FUNCTION_BLOCK WoodBunkEx EXTENDS SectionEx
VAR //references to objects imported from Hardware GVL - using references instead of VAR_EXTERNAL or direct access allows local renaming
	robotLeft, robotRight : REFERENCE TO Robot;
	
	stagingTableLeft, stagingTableRight : REFERENCE TO WoodBunkTable;
	magazineLeft, magazineRight: REFERENCE TO MaterialStorage;
	
	strapper : REFERENCE TO StrapMachine;
	
	insertionLeft, insertionRight : REFERENCE TO Insertion;
	insertionBottom : REFERENCE TO AirPiston;
	
	toolStorageLeft, toolStorageRight : REFERENCE TO A21ToolStorage;
END_VAR
VAR
	conveyorPos : REAL;
	
	insertionSlots : ARRAY[Surface.TOP..Surface.BOTTOM] OF STRING;
	
	materialsArr : POINTER TO PositionMaterials; //array of PositionMaterials
	currentPair : REFERENCE TO PositionMaterials;
	
	stagingMaterial : STRING; //ex: currentPair.left
	currentMaterial : STRING; //ex: WDS18_WDS20 --> WDS18, then WDS20
	
	stagingTemplateReady : BOOL;
	stagingTemplateLeft : WoodBunkTable;
	stagingTemplateRight : WoodBunkTable;
	
	step : (RUN_TO_POSITION, PUSH, RUN_TO_STRAP, STRAP, RELEASE, RESET);
	
	//for staging use
	stageSet : INT;	
	stageStepLeft, stageStepRight : INT;
	iStagingSlotLeft, iStagingSlotRight : INT;
	
	robotLeftOutputs, robotRightOutputs : ARRAY[1..50] OF INT;
END_VAR
VAR
	tempInspectionSuite : VisionSuite; //send/receive from TcpServer
	leftInspectionFrame, rightInspectionFrame : VisionFrame; //parsed from above
END_VAR
VAR CONSTANT
	leftCamera : INT := 1;
	rightCamera : INT := 2;
END_VAR

entryRefPos := conveyorPos;
exitRefPos := conveyorPos;

SUPER^();

CASE status OF
	SectionStatus.IDLE:
		//RETURN;
	
	SectionStatus.ALIGNING:
		//
		
	SectionStatus.ACTIVE:
		//
		
	SectionStatus.CLEARING:
		stagingTemplateReady := FALSE;
		
	SectionStatus.COMPLETE:	
		//
		
	-100:
		RETURN;
		
END_CASE

materialsArr := ADR(currentBundle.woodBunk);

loaded := 
	insertionSlots[Surface.TOP] = materialsArr[iPair].top AND
	insertionSlots[Surface.LEFT] = materialsArr[iPair].left AND
	insertionSlots[Surface.RIGHT] = materialsArr[iPair].right AND
	insertionSlots[Surface.BOTTOM] = materialsArr[iPair].bottom;
	
//bundle needs this section's materials, and either robot failed
IF usesProcess() AND NOT(robotLeft.operational AND robotRight.operational) THEN 

	currentBypass := TRUE;
	RETURN;
END_IF //otherwise, carry over bypass from prev section

stage();

METHOD changeRobotsEOAT : BOOL
VAR_INPUT
END_VAR
IF robotLeft.tool <> sectionID THEN
	MEMSET(ADR(robotLeftOutputs), 0, SIZEOF(robotLeftOutputs));
	robotLeftOutputs[1] := A21.TOOL_CHANGE_CHIPBOARD;
	robotLeft.setParamsAndWait(robotLeftOutputs);
END_IF

IF robotRight.tool <> sectionID THEN
	MEMSET(ADR(robotRightOutputs), 0, SIZEOF(robotRightOutputs));
	robotRightOutputs[1] := A21.TOOL_CHANGE_CHIPBOARD;
	robotRight.setParamsAndWait(robotRightOutputs);
END_IF

changeRobotsEOAT := robotLeft.tool = sectionID AND robotRight.tool = sectionID;
END_METHOD

METHOD PROTECTED createStagingTemplate : BOOL
VAR
	remainingMaterial : STRING;
	splitMaterial : STRING;
	
	i : INT;
END_VAR
FOR i:=0 TO GVL.maxPairs BY 1 DO //iterate through all pairs and autofill the template
	//LEFT TABLE
	remainingMaterial := materialsArr[i].top;
	WHILE FIND(remainingMaterial, '_') > 0 DO //until no underscore found
		splitCombinedMaterials(remainingMaterial, splitMaterial);
		stagingTemplateLeft.autofill(splitMaterial);
	END_WHILE
	stagingTemplateLeft.autofill(remainingMaterial);
	
	remainingMaterial := materialsArr[i].left;
	WHILE FIND(remainingMaterial, '_') > 0 DO
		splitCombinedMaterials(remainingMaterial, splitMaterial);
		stagingTemplateLeft.autofill(splitMaterial);
	END_WHILE
	stagingTemplateLeft.autofill(remainingMaterial);
	
	//RIGHT TABLE
	remainingMaterial := materialsArr[i].right;
	WHILE FIND(remainingMaterial, '_') > 0 DO
		splitCombinedMaterials(remainingMaterial, splitMaterial);
		stagingTemplateRight.autofill(splitMaterial);
	END_WHILE
	stagingTemplateRight.autofill(remainingMaterial);
	
	remainingMaterial := materialsArr[i].bottom;
	WHILE FIND(remainingMaterial, '_') > 0 DO
		splitCombinedMaterials(remainingMaterial, splitMaterial);
		stagingTemplateRight.autofill(splitMaterial);
	END_WHILE
	stagingTemplateRight.autofill(remainingMaterial);
END_FOR
END_METHOD

METHOD findOpenSlot : BOOL
VAR_INPUT
	materialCode : STRING;
END_VAR
VAR_OUTPUT
	openSlot : INT := 0;
END_VAR
(*
IF FIND(materialCode, 'WDW') > 0 THEN //top wide, load in slot 0-1
	FOR i:=1 TO 2 BY 1 DO
		IF stageTableLeft[i] = '' THEN
			findOpenSlot := TRUE;
			openSlot := i;
			RETURN;
		END_IF
	END_FOR
	
ELSIF FIND(materialCode, 'WDT') > 0 OR FIND(materialCode, 'WDS') > 0 THEN //top std and sides, load in slot 2-9
	FOR i:=3 TO 10 BY 1 DO
		IF stageTableLeft[i] = '' THEN
			findOpenSlot := TRUE;
			openSlot := i;
			RETURN;
		END_IF
	END_FOR
	
END_IF
*)
END_METHOD

METHOD initHardware : BOOL
conveyors := ADR(allConveyors);

robotLeft REF= robots[1];
robotRight REF= robots[2];

strapper REF= strapperA21;

insertionLeft REF= insertionA21Left;
insertionLeft REF= insertionA21Right;

stagingTableLeft REF= stagingTableLeft;
stagingTableRight REF= stagingTableRight;

magazineLeft REF= woodBunkMagazineLeft;
magazineRight REF= woodBunkMagazineRight;

(*
strapper REF= Hardware.strapper;

insertionLeft REF= Hardware.insertionWoodBunkSides[Surface.LEFT];
insertionLeft REF= Hardware.insertionWoodBunkSides[Surface.RIGHT];

stagingTableLeft REF= Hardware.stagingTable[Surface.LEFT];
stagingTableRight REF= Hardware.stagingTable[Surface.RIGHT];

magazineLeft REF= Hardware.woodBunkMagazine[Surface.LEFT];
magazineRight REF= Hardware.woodBunkMagazine[Surface.RIGHT];
*)
END_METHOD

METHOD PROTECTED load : BOOL
VAR_INPUT
	pair : REFERENCE TO PositionMaterials;
END_VAR
IF NOT robotLeft.operational OR NOT robotLeft.operational THEN
	error := TRUE;
	
	currentBypass := TRUE;
	RETURN;
END_IF

IF NOT (robotLeft.reserve(sectionID) AND robotRight.reserve(sectionID)) THEN
	RETURN;
END_IF

IF NOT (robotLeft.tool = sectionID AND robotRight.tool = sectionID) THEN //robots have wrong tool
	changeRobotsEOAT(); //wait for robots to finish changing tools
	RETURN;
END_IF


CASE loadSet OF
	0: //top and bottom
		IF 
			loadingSequence(
				actingRobot:= robotLeft, 
				robotOutputs:= robotLeftOutputs, 
				stagingTable:= stagingTableLeft, 
				loadStep:= loadStepLeft, 
				surfaceID:= Surface.TOP, 
				material:= pair.top, 
				fail=> )
			AND
			loadingSequence(
				actingRobot:= robotRight, 
				robotOutputs:= robotRightOutputs, 
				stagingTable:= stagingTableRight, 
				loadStep:= loadStepRight, 
				surfaceID:= Surface.BOTTOM, 
				material:= pair.bottom, 
				fail=> )
		THEN
			loadStepLeft := loadStepRight := 0;
			loadSet := 10;
		END_IF
		
	10: //sides
		IF
			loadingSequence(
				actingRobot:= robotLeft, 
				robotOutputs:= robotLeftOutputs, 
				stagingTable:= stagingTableLeft, 
				loadStep:= loadStepLeft, 
				surfaceID:= Surface.LEFT, 
				material:= pair.left, 
				fail=> )
			AND
			loadingSequence(
				actingRobot:= robotRight, 
				robotOutputs:= robotRightOutputs, 
				stagingTable:= stagingTableRight, 
				loadStep:= loadStepRight, 
				surfaceID:= Surface.RIGHT, 
				material:= pair.right, 
				fail=> )
		THEN
			loadStepLeft := loadStepRight := 0;
			loadSet := COMPLETE;
		END_IF
		
	COMPLETE:
		loadSet := 0;
		loadStepLeft := loadStepRight := 0;
		
		loaded := 
			insertionSlots[Surface.TOP] = materialsArr[iPair].top AND
			insertionSlots[Surface.LEFT] = materialsArr[iPair].left AND
			insertionSlots[Surface.RIGHT] = materialsArr[iPair].right AND
			insertionSlots[Surface.BOTTOM] = materialsArr[iPair].bottom;
		
		robotLeft.release(sectionID);
		robotRight.release(sectionID);
		
		load := TRUE;
END_CASE
END_METHOD

METHOD loadBottom : BOOL
VAR_IN_OUT //acting refers to which robot is performing the task, if the designated robot fails the other may take over
	actingRobot : Robot;
	robotOutputs : ARRAY[1..50] OF INT;
	actingStagingTable : WoodBunkTable;
	actingLoadStep : INT;
END_VAR
VAR_INPUT
	material : STRING;
END_VAR
VAR_OUTPUT
	fail : BOOL;
END_VAR
VAR
	slot : INT;
END_VAR
IF
	actingLoadStep <> COMPLETE AND_THEN
	NOT actingRobot.reserve(sectionID)
THEN
	RETURN;
END_IF

CASE actingLoadStep OF
	0:
		IF NOT actingStagingTable.findSlot(materialID := material, atSlot => slot) THEN
			fail := TRUE;
			RETURN;
		END_IF
		
		MEMSET(ADR(robotOutputs), 0, SIZEOF(robotOutputs));
		robotOutputs[1] := A21.LOAD_BUNK_TO_BOTTOM;
		robotOutputs[2] := slot;
		
		IF actingRobot.setParamsAndWait(robotOutputs) THEN
			actingLoadStep := COMPLETE;
		END_IF
		
	COMPLETE:
		//turn suction on
		actingRobot.release(sectionID);
		loadBottom := TRUE;
END_CASE
END_METHOD

METHOD loadingSequence : BOOL
VAR_IN_OUT
	actingRobot : Robot;
	robotOutputs : ARRAY[1..50] OF INT;
	stagingTable : WoodBunkTable;
	loadStep : INT;
END_VAR
VAR_INPUT
	surfaceID : Surface;
	material : STRING;
END_VAR
VAR_OUTPUT
	fail : BOOL;
END_VAR
VAR
	slot : INT;
END_VAR
IF material = '' THEN
	loadingSequence := TRUE;
	RETURN;
END_IF

CASE loadStep OF
	0:
		IF NOT stagingTable.findSlot(materialID := material, atSlot => slot) THEN
			fail := TRUE;
			RETURN;
		END_IF
		
		MEMSET(ADR(robotOutputs), 0, SIZEOF(robotOutputs));
		CASE surfaceID OF
			Surface.TOP: 					robotOutputs[1] := A21.LOAD_BUNK_TO_TOP;
			Surface.LEFT, Surface.RIGHT: 	robotOutputs[1] := A21.LOAD_BUNK_TO_SIDE;
			Surface.BOTTOM: 				robotOutputs[1] := A21.LOAD_BUNK_TO_BOTTOM;
		END_CASE
		robotOutputs[2] := slot;
		
		IF actingRobot.setParamsAndWait(robotOutputs) THEN
			loadStep := COMPLETE;
		END_IF
		
	COMPLETE:
		//turn suction on
		actingRobot.release(sectionID);
		loadingSequence := TRUE;
		
END_CASE
END_METHOD

METHOD loadSides : BOOL
VAR_IN_OUT //acting refers to which robot is performing the task, if the designated robot fails the other may take over
	actingRobot : Robot;
	robotOutputs : ARRAY[1..50] OF INT;
	actingStagingTable : WoodBunkTable;
	actingLoadStep : INT;
END_VAR
VAR_INPUT
	material : STRING;
END_VAR
VAR_OUTPUT
	fail : BOOL;
END_VAR
VAR
	slot : INT;
END_VAR
IF
	actingLoadStep <> COMPLETE AND_THEN
	NOT actingRobot.reserve(sectionID)
THEN
	RETURN;
END_IF

CASE actingLoadStep OF
	0:
		IF NOT actingStagingTable.findSlot(materialID := material, atSlot => slot) THEN
			fail := TRUE;
			RETURN;
		END_IF
		
		MEMSET(ADR(robotOutputs), 0, SIZEOF(robotOutputs));
		robotOutputs[1] := A21.LOAD_BUNK_TO_SIDE;
		robotOutputs[2] := slot;
		
		IF actingRobot.setParamsAndWait(robotOutputs) THEN
			actingLoadStep := COMPLETE;
		END_IF
		
	COMPLETE:
		//turn suction on
		actingRobot.release(sectionID);
		loadSides := TRUE;
END_CASE
END_METHOD

METHOD loadTop : BOOL
VAR_IN_OUT //acting refers to which robot is performing the task, if the designated robot fails the other may take over
	actingRobot : Robot;
	robotOutputs : ARRAY[1..50] OF INT;
	actingStagingTable : WoodBunkTable;
	actingLoadStep : INT;
END_VAR
VAR_INPUT
	material : STRING;
END_VAR
VAR_OUTPUT
	fail : BOOL;
END_VAR
VAR
	slot : INT;
END_VAR
IF
	actingLoadStep <> COMPLETE AND_THEN
	NOT actingRobot.reserve(sectionID)
THEN
	RETURN;
END_IF

CASE actingLoadStep OF
	0:
		IF NOT actingStagingTable.findSlot(materialID := material, atSlot => slot) THEN
			fail := TRUE;
			RETURN;
		END_IF
		
		MEMSET(ADR(robotOutputs), 0, SIZEOF(robotOutputs));
		robotOutputs[1] := A21.LOAD_BUNK_TO_TOP;
		robotOutputs[2] := slot;
		
		IF actingRobot.setParamsAndWait(robotOutputs) THEN
			actingLoadStep := COMPLETE;
		END_IF
		
	COMPLETE:
		//turn suction on
		actingRobot.release(sectionID);
		loadTop := TRUE;
END_CASE
END_METHOD

METHOD PROTECTED process : BOOL
VAR
	currentPair : REFERENCE TO PositionMaterials REF= materialsArr[iPair];
END_VAR
IF iPair >= GVL.maxPairs THEN
	process := TRUE;
	RETURN;
END_IF

IF NOT PositionIsValid(pair:= currentPair) THEN
	step := 0;
	iPair := iPair + 1;
	RETURN;
END_IF

CASE step OF
	RUN_TO_POSITION: //free run until position reached
		IF directionCheckAndSet(conveyorPos, currentPair.position) AND load(pair:= currentPair) THEN
			step := PUSH;
		END_IF

	PUSH: //push command
		setConveyorMode(ConveyorMode.STOP);
		IF
			NOT insertionLeft.align(currentBundle.height/2) OR
			NOT insertionRight.align(currentBundle.height/2)
		THEN
			RETURN;
		END_IF
		
		insertionLeft.press();
		insertionRight.press();
		insertionBottom.extend();
		
		IF insertionLeft.contact AND insertionRight.contact AND insertionBottom.contact THEN		
			step := STRAP;
		END_IF
		
	STRAP: //strap command
		//turn off suction here
		setConveyorMode(ConveyorMode.STOP);
		IF strapper.ready OR (NOT strapper.busy AND NOT strapper.error) THEN
			strapper.strap();
		END_IF
		
		IF strapper.done THEN
			step := RELEASE;
		END_IF
		
	RELEASE: //release command
		setConveyorMode(ConveyorMode.STOP);
		
		IF NOT insertionLeft.home THEN
			insertionLeft.align(0);
			insertionLeft.release();
		END_IF
		
		IF NOT insertionRight.home THEN
			insertionRight.align(0);
			insertionRight.release();
		END_IF
		
		IF insertionLeft.home AND insertionRight.home THEN
			step := RESET;
		END_IF
		
	RESET: //reset
		setConveyorMode(ConveyorMode.FORWARD);
		iPair := iPair + 1;
		
		step := 0;
		
END_CASE
END_METHOD

METHOD splitCombinedMaterials : BOOL
VAR_IN_OUT
	materialID : STRING;
	splitMaterial : STRING;
END_VAR
VAR
	i : INT;
END_VAR
FindAndSplitChar(
	sSeparatorChar:= '_', 
	pSrcString:= ADR(materialID), 
	pLeftString:= ADR(splitMaterial), 
	nLeftSize:= SIZEOF(splitMaterial), 
	pRightString:= ADR(materialID), 
	nRightSize:= SIZEOF(materialID), 
	bSearchFromRight:= FALSE);
END_METHOD

METHOD stage : BOOL
//robot reservation needs to be constantly checked so it is not in the state machine
IF NOT (robotLeft.reserve(sectionID) AND robotRight.reserve(sectionID)) THEN
	RETURN;
END_IF

IF NOT (robotLeft.tool = sectionID AND robotRight.tool = sectionID) THEN //robots have wrong tool
	changeRobotsEOAT(); //wait for robots to finish changing tools
	RETURN;
END_IF

CASE stageSet OF
	0: //create staging template
		createStagingTemplate();
		stageSet := 10;
	
	10: //staging sequence
		IF TcpServer1Vision.fetch(tempInspectionSuite.data) THEN
			(*
				1 - parse
				2 - determine if the camera number is for left or right staging
				3 - copy into appropriate frame
			*)
			MEMCPY(
				ADR(tempInspectionSuite.json),
				ADR(tempInspectionSuite.data),
				MIN( SIZEOF(tempInspectionSuite.json), SIZEOF(tempInspectionSuite.data) ));
			
			VisionJsonParser(
				jsonString:= tempInspectionSuite.json,
				visionData=> );
			
			IF NOT FrameIsValid(tempInspectionSuite.frame) THEN
				//
			
			ELSIF tempInspectionSuite.frame.CameraNumber = leftCamera THEN
				leftInspectionFrame := tempInspectionSuite.frame;
				
			ELSIF tempInspectionSuite.frame.CameraNumber = rightCamera THEN
				rightInspectionFrame := tempInspectionSuite.frame;
				
			END_IF
		END_IF
		

		IF
			stagingSequence(
				template:= stagingTemplateLeft, 
				magazine:= magazineLeft, 
				table:= stagingTableLeft, 
				stagingSlot:= iStagingSlotLeft,
				actingRobot:= robotLeft, 
				robotOutputs:= robotLeftOutputs,
				inspectionFrame:= leftInspectionFrame, 
				actingStep:= stageStepLeft, 
				camera:= leftCamera, 
				fail=> )
			AND
			stagingSequence(
				template:= stagingTemplateRight, 
				magazine:= magazineRight, 
				table:= stagingTableRight, 
				stagingSlot:= iStagingSlotRight,
				actingRobot:= robotRight, 
				robotOutputs:= robotRightOutputs,
				inspectionFrame:= rightInspectionFrame, 
				actingStep:= stageStepRight, 
				camera:= rightCamera, 
				fail=> )
		THEN
			stageStepLeft := stageStepRight := 0;
			iStagingSlotLeft := iStagingSlotRight := 0;
			
			stageSet := COMPLETE;
		END_IF
		
	COMPLETE:
		stageSet := 0;
		stageStepLeft := stageStepRight := 0;
		
		robotLeft.release(sectionID);
		robotRight.release(sectionID);
		
		stage := TRUE;
		
END_CASE
END_METHOD

METHOD stageLeft : BOOL
VAR_IN_OUT
	template : WoodBunkTable;
	magazine : MaterialStorage;
	table : WoodBunkTable;
	actingStagingSlot : INT;
	actingRobot : Robot;
	robotOutputs : ARRAY[1..50] OF INT;
	actingFrame : VisionFrame;
	actingStep : INT;
END_VAR
VAR_INPUT
	camera : INT;
END_VAR
VAR_OUTPUT
	fail : BOOL;
END_VAR
VAR
	finished : BOOL;
	slot : INT;
	templateArr : POINTER TO STRING;
END_VAR
VAR CONSTANT
	WIP : INT := 0;
	PASSED : INT := 1;
	FAILED : INT := 2;
END_VAR
IF table.isFull() OR actingStagingSlot > 10 THEN
	stageLeft := TRUE;
	RETURN;
END_IF

templateArr := template.getSlotsAsArray();

//follow the template as is
IF NOT magazine.findSlot(materialID:= templateArr[actingStagingSlot], atSlot => slot) THEN
	fail := TRUE;
	RETURN;
END_IF

IF actingStep > 0 THEN
	finished := actingRobot.setCommandAndWait(A21.STAGE_BUNK, slot, actingStagingSlot, 0);
END_IF

CASE actingStep OF
	0: //command
		IF actingRobot.inputs[5].10 THEN
			actingStep := 10;
		END_IF
		
	10: //request inspection
		tempInspectionSuite.frame.MaterialID := templateArr[actingStagingSlot];
		tempInspectionSuite.frame.CheckFor := 'ORIENTATION';
		tempInspectionSuite.frame.CameraNumber := camera;
	
		CreateJsonDocumentAuto(
			visionFrameData:= tempInspectionSuite.frame, 
			jsonDocument=> tempInspectionSuite.json);
		
		MEMCPY(
			ADR(tempInspectionSuite.data), 
			ADR(tempInspectionSuite.json), 
			MIN( SIZEOF(tempInspectionSuite.data), SIZEOF(tempInspectionSuite.json) ));
			
		TcpServer1Vision.queue(tempInspectionSuite.data);
		
		actingStep := 20;
	
	20: //fetch inspection data and parse
		actingRobot.setCommandAndWait(A21.STAGE_BUNK, slot, actingStagingSlot, 0);
		robotOutputs[4] := 0;
		
		IF NOT FrameIsValid(actingFrame) THEN
			RETURN;
		END_IF
		
		IF actingFrame.SuccessFlag = 1 THEN
			robotOutputs[4] := PASSED;
		ELSE
			robotOutputs[4] := FAILED;
		END_IF
		actingStep := 30;
		
	30: //finish command
		IF finished THEN
			IF actingFrame.SuccessFlag = 1 THEN
				actingStagingSlot := actingStagingSlot + 1;
			END_IF
			
			actingStep := 0;
		END_IF
END_CASE
END_METHOD

METHOD stageRight : BOOL
VAR_IN_OUT
	template : WoodBunkTable;
	magazine : MaterialStorage;
	table : WoodBunkTable;
	actingStagingSlot : INT;
	actingRobot : Robot;
	actingFrame : VisionFrame;
	actingStep : INT;
END_VAR
VAR_INPUT
	camera : INT;
END_VAR
VAR_OUTPUT
	fail : BOOL;
END_VAR
VAR
	finished : BOOL;
	robotOutputs : POINTER TO INT;
	
	slot : INT;
	templateArr : POINTER TO STRING;
	
END_VAR
IF table.isFull() OR actingStagingSlot > 10 THEN
	stageRight := TRUE;
	RETURN;
END_IF

templateArr := template.getSlotsAsArray();

//follow the template as is
IF NOT magazine.findSlot(materialID:= templateArr[actingStagingSlot], atSlot => slot) THEN
	fail := TRUE;
	RETURN;
END_IF

IF actingStep > 0 THEN
	finished := actingRobot.setCommandAndWait(A21.STAGE_BUNK, slot, actingStagingSlot, 0);
END_IF

CASE actingStep OF
	0: //command
		IF actingRobot.inputs[5].10 THEN
			actingStep := 10;
		END_IF
		
	10: //send inspection data
		tempInspectionSuite.frame.MaterialID := templateArr[actingStagingSlot];
		tempInspectionSuite.frame.CheckFor := 'ORIENTATION';
		tempInspectionSuite.frame.CameraNumber := camera;
	
		CreateJsonDocumentAuto(
			visionFrameData:= tempInspectionSuite.frame, 
			jsonDocument=> tempInspectionSuite.json);
		
		MEMCPY( //data = json
			ADR(tempInspectionSuite.data), 
			ADR(tempInspectionSuite.json), 
			MIN( SIZEOF(tempInspectionSuite.data), SIZEOF(tempInspectionSuite.json) ));
			
		TcpServer1Vision.queue(tempInspectionSuite.data);
		
		actingStep := 20;
	
	20: //fetch inspection data and parse
		actingRobot.setCommandAndWait(A21.STAGE_BUNK, slot, actingStagingSlot, 0);
		robotOutputs[11] := 0;
		
		IF NOT FrameIsValid(actingFrame) THEN
			RETURN;
		END_IF
		
		IF actingFrame.SuccessFlag = 1 THEN
			robotOutputs[11] := 1;
		ELSE
			robotOutputs[11] := 2;
		END_IF
		actingStep := 30;
		
	30: //finish command
		IF finished THEN
			IF actingFrame.SuccessFlag = 1 THEN
				actingStagingSlot := actingStagingSlot + 1;
			END_IF
			
			actingStep := 0; //stage next
		END_IF
		
END_CASE
END_METHOD

METHOD stagingSequence : BOOL
VAR_IN_OUT
	template : WoodBunkTable;
	magazine : MaterialStorage;
	table : WoodBunkTable;
	stagingSlot : INT;
	actingRobot : Robot;
	robotOutputs : ARRAY[1..50] OF INT;
	inspectionFrame : VisionFrame;
	actingStep : INT;
END_VAR
VAR_INPUT
	camera : INT;
END_VAR
VAR_OUTPUT
	fail : BOOL;
END_VAR
VAR
	finished : BOOL;
	slot : INT;
	templateArr : POINTER TO STRING;
END_VAR
VAR CONSTANT
	WIP : INT := 0;
	PASSED : INT := 1;
	FAILED : INT := 2;
END_VAR
IF table.isFull() OR stagingSlot > 10 THEN
	stagingSequence := TRUE;
	RETURN;
END_IF

templateArr := template.getSlotsAsArray();

//follow the template as is
IF NOT magazine.findSlot(materialID:= templateArr[stagingSlot], atSlot => slot) THEN
	fail := TRUE;
	RETURN;
END_IF

IF actingStep > 0 THEN
	finished := actingRobot.setCommandAndWait(A21.STAGE_BUNK, slot, stagingSlot, 0);
END_IF

CASE actingStep OF		
	0: //command
		IF actingRobot.inputs[5].10 THEN
			actingStep := 10;
		END_IF
		
	10: //request inspection
		tempInspectionSuite.frame.MaterialID := templateArr[stagingSlot];
		tempInspectionSuite.frame.CheckFor := 'ORIENTATION';
		tempInspectionSuite.frame.CameraNumber := camera;
	
		CreateJsonDocumentAuto(
			visionFrameData:= tempInspectionSuite.frame, 
			jsonDocument=> tempInspectionSuite.json);
		
		MEMCPY(
			ADR(tempInspectionSuite.data), 
			ADR(tempInspectionSuite.json), 
			MIN( SIZEOF(tempInspectionSuite.data), SIZEOF(tempInspectionSuite.json) ));
			
		TcpServer1Vision.queue(tempInspectionSuite.data);
		
		actingStep := 20;
	
	20: //fetch inspection data and parse
		actingRobot.setCommandAndWait(A21.STAGE_BUNK, slot, stagingSlot, 0);
		robotOutputs[4] := 0;
		
		IF NOT FrameIsValid(inspectionFrame) THEN
			RETURN;
		END_IF
		
		IF inspectionFrame.SuccessFlag = 1 THEN
			robotOutputs[4] := PASSED;
		ELSE
			robotOutputs[4] := FAILED;
		END_IF
		actingStep := 30;
		
	30: //finish command
		IF finished THEN
			IF inspectionFrame.SuccessFlag = 1 THEN
				stagingSlot := stagingSlot + 1;
			END_IF
			
			actingStep := 0;
		END_IF
END_CASE
END_METHOD

METHOD PROTECTED usesProcess : BOOL
VAR
	i : INT;
END_VAR
IF materialsArr = 0 THEN
	RETURN;
END_IF

FOR i:=0 TO GVL.maxPairs BY 1 DO
	IF PositionIsValid(materialsArr[i]) THEN
		usesProcess := TRUE;
		RETURN;
	END_IF
END_FOR
END_METHOD

END_FUNCTION_BLOCK

(* stored: Version 1.1.0.1, ProductVersion 3.1.4024.11
   POU WoodBunkEx: Id {2aa6527c-a14c-44cf-be9f-979ab3b36650}, SpecialFunc None
   Folder Helper: Id {0ee277a5-addc-4b61-878e-d1cc157f6dd0}
   Folder Loading: Id {0eb4d7b4-792d-4f5b-94c4-a31b58b4e298}
   Folder Staging: Id {bc681162-e30f-4f50-871c-01b6e331ef41}
   Folder z_Obsolete: Id {dd13f688-1c3e-407f-adbc-850fb11e2559}
   Method changeRobotsEOAT: Id {0175a478-48f8-4f51-9aaa-685d24fb2e12}
   Method createStagingTemplate: Id {8e787035-737c-49d2-b5f7-4777f799dafd}
   Method findOpenSlot: Id {2a2b3fd4-a6db-4ee8-9905-0e408a84c931}
   Method initHardware: Id {6f231511-302e-4630-b885-f7ba64cde469}
   Method load: Id {92ab4615-f272-434d-9633-4b50d2b91dde}
   Method loadBottom: Id {73f10a94-e5aa-4e92-97d8-a569974a35c3}
   Method loadingSequence: Id {227dbd1b-1079-40ed-96b7-116088e0949c}
   Method loadSides: Id {3ccf08fc-463f-49c8-8c1d-2d0486dfc15c}
   Method loadTop: Id {07f819a0-292a-4f85-a714-fbbd36b2c69a}
   Method process: Id {597597cf-314e-4ce5-b2f7-4e1ca8bb518a}
   Method splitCombinedMaterials: Id {6e69d6d2-13f5-49f2-80c0-511c5addb1ee}
   Method stage: Id {e862c418-7b88-460a-9fd6-b732a3ca8dda}
   Method stageLeft: Id {c5da086f-368a-4e05-be45-9cffdf019f3a}
   Method stageRight: Id {23be37a6-4be3-40ad-b42f-0243ecc2653b}
   Method stagingSequence: Id {5bc1d781-6d11-4e38-87a4-80c150730fb1}
   Method usesProcess: Id {b0bfdc8e-1617-46c3-aaf0-1372637d9607} *)
